Universal Robots PolyScope program: L06_extract_force.urp

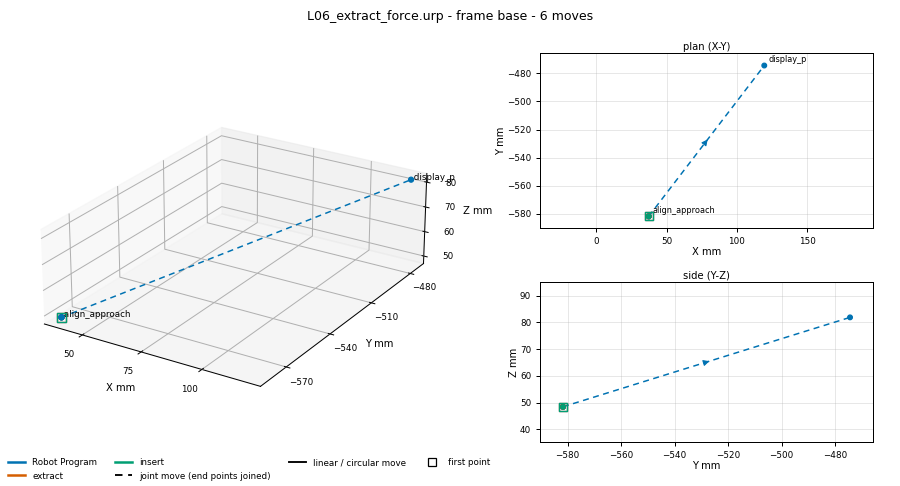
[picture p0: tool path of L06_extract_force.urp in frame base, 6 of 8 moves have a stored position in this frame; points joined in program order, loops and branches not executed]
Program L06_extract_force (installation=default directory=/programs createdIn=5.9.1.1031110 lastSavedIn=5.9.1.1031110 robotSerialNumber=20195501059)
Calibrated DH parameters: a=[0.000146, -0.418764, -0.053981, 0.000058, -0.000023, 0]; d=[0.162545, 37.319448, -206.067439, 168.881546, 0.09955, 0.099464]; alpha=[1.57004, -0.001979, 0.002304, 1.570607, -1.57066, 0]; deltaTheta=[0, -0.174616, -1.258233, 1.432844, -0.000001, 0]
BeforeStart
  URCap Gripper Activate (Robotiq_Grippers, Robotiq Inc.) dataModel(ResetAndActivateKey=false)
  URCap Gripper (Robotiq_Grippers, Robotiq Inc.) dataModel(position=60.0, force=10.0, speed=40.0, positionInDouble=60.0, forceInDouble=10.0, speedInDouble=40.0, slaveIds=[9], blocking=true)
  start_p := get_actual_tcp_pose()
  MoveJ speed 60 deg/s, acceleration 80 deg/s^2 (useActiveTCP=true) feature=Base
    Waypoint Waypoint (Variable): variable=start_p
  MoveL speed 250 mm/s, acceleration 1200 mm/s^2 (useActiveTCP=true) feature=Base
    MoveDirectionNode (selectedDirection=ZPlus)
      Until DISTANCE (allowActions=false deceleration=3 distanceNodeType=STOP) Distance=0.025; motionParameters(blendRadius=0)
  URCap Gripper (Robotiq_Grippers, Robotiq Inc.) dataModel(position=100.0, force=25.0, speed=100.0, positionInDouble=100.0, forceInDouble=25.0, speedInDouble=100.0, slaveIds=[9], blocking=true)
Robot Program (runOnlyOnce=true)
  MoveJ speed 60 deg/s, acceleration 80 deg/s^2 (useActiveTCP=true) feature=Base
    Waypoint align_approach: TCP in base x=37.324 y=-581.757 z=48.473 mm, rx=2.21 ry=2.2328 rz=0 rad; joints [80.399, -68.66, 105.716, -127.049, 270.027, 79.839] deg; TCP offset x=0 y=0 z=174 mm, rx=0 ry=0 rz=0 rad
  MoveL speed 250 mm/s, acceleration 1200 mm/s^2 (useActiveTCP=true) feature=Base
    Waypoint misalign: TCP in base x=37.345 y=-581.767 z=48.476 mm, rx=2.3536 ry=2.027 rz=0.0112 rad; joints [79.512, -69.245, 106.923, -128.62, 271.871, 88.086] deg
    'Touch plug'
    URCap Gripper (Robotiq_Grippers, Robotiq Inc.) dataModel(position=100.0, force=25.0, speed=100.0, positionInDouble=100.0, forceInDouble=25.0, speedInDouble=100.0, slaveIds=[9], blocking=true)
    MoveDirectionNode (selectedDirection=ZPlus toolParams=0.02, 0.8) feature=Joint_6_name
      Until DISTANCE (allowActions=true deceleration=3 distanceNodeType=STOP) Distance=0.025; motionParameters(blendRadius=0)
        MoveL speed 250 mm/s, acceleration 1200 mm/s^2 (useActiveTCP=true) feature=Base
          Waypoint align_approach: TCP in base x=37.324 y=-581.757 z=48.473 mm, rx=2.21 ry=2.2328 rz=0 rad; joints [80.399, -68.66, 105.716, -127.049, 270.027, 79.839] deg
          Halt
      Until TOOL_CONTACT_DETECTION (allowActions=false retraction=0.002 decelerationAcceleration=0.8 decelerationAngularAcceleration=34.906585)
    Call extract
    extract_p := get_actual_tcp_pose()
    MoveDirectionNode (selectedDirection=YPlus) feature=Base
      Until DISTANCE (allowActions=false deceleration=3 distanceNodeType=STOP) Distance=0.05; motionParameters(blendRadius=0)
    MoveJ speed 60 deg/s, acceleration 80 deg/s^2 (useActiveTCP=true) feature=Base
      Waypoint display_p: TCP in base x=119.536 y=-474.453 z=81.895 mm, rx=0.3577 ry=2.5974 rz=0.0553 rad; joints [71.361, -83.619, 123.353, -121.111, 298.741, -5.14] deg
      Wait Sleep waitTime=2
      Waypoint Waypoint (Variable): variable=extract_p
    'Deliberately misalign'
    MoveDirectionNode (selectedDirection=ZPlus) feature=Joint_6_name
      Until DISTANCE (allowActions=false deceleration=3 distanceNodeType=STOP) Distance=0.001; motionParameters(blendRadius=0)
    MoveDirectionNode (selectedDirection=XPlus) feature=Joint_6_name
      Until DISTANCE (allowActions=false deceleration=3 distanceNodeType=STOP) Distance=0.001; motionParameters(blendRadius=0)
    Call insert
SubProgram -> insert
SubProgram -> extract
SubProgram extract (keepSynchronizedWithDisk=false)
  MoveL speed 250 mm/s, acceleration 1200 mm/s^2 (useActiveTCP=true) feature=Base
    URCap Gripper (Robotiq_Grippers, Robotiq Inc.) dataModel(position=60.0, force=100.0, speed=100.0, positionInDouble=60.0, forceInDouble=100.0, speedInDouble=100.0, slaveIds=[9], blocking=true)
    MoveDirectionNode (selectedDirection=ZMinus)
      Until DISTANCE (allowActions=false deceleration=3 distanceNodeType=STOP) Distance=0.02; motionParameters(blendRadius=0)
    URCap Zero FT Sensor (Robotiq_Copilot, Robotiq Inc.) dataModel(NodeInitializedKey=true, WaitForSteadyWrenchOptionKey=true)
    URCap Gripper (Robotiq_Grippers, Robotiq Inc.) dataModel(position=100.0, force=25.0, speed=100.0, positionInDouble=100.0, forceInDouble=25.0, speedInDouble=100.0, slaveIds=[9], blocking=true)
    URCap Grip Check (Robotiq_Grippers, Robotiq Inc.) dataModel(ObjectDetectedKey=true, DimensionValidationKey=false, DimensionKey=100.0, DimensionDimensionPositiveGapKey=5.0, DimensionNegativeGapKey=5.0, GripperIdKey=1, ModelDefinedKey=true); state(isChildrenLocked=true)
      URCap If (Robotiq_Grippers, Robotiq Inc.)
        'plug grabbed'
      URCap Else (Robotiq_Grippers, Robotiq Inc.)
        'no plug'
        MoveJ speed 60 deg/s, acceleration 80 deg/s^2 (useActiveTCP=true) feature=Base
          Waypoint align_approach: TCP in base x=37.324 y=-581.757 z=48.473 mm, rx=2.21 ry=2.2328 rz=0 rad; joints [80.399, -68.66, 105.716, -127.049, 270.027, 79.839] deg
          Halt
    'Let gripper seek alignment'
    URCap Force Control (Robotiq_Copilot, Robotiq Inc.) dataModel(NodeInitializedKey=true, force_x=0, force_y=0, force_z=0, force_mx=0, force_my=0, force_mz=0, limit_x_neg=-100, limit_y_neg=-100, limit_z_neg=-100, limit_x_pos=100, limit_y_pos=100, limit_z_pos=100, limit_mx_neg=-20, limit_my_neg=-20, limit_mz_neg=-20, limit_mx_pos=20, limit_my_pos=20, limit_mz_pos=20, stiffness_x=100, stiffness_y=100, stiffness_z_position=100, stiffness_mx=100, stiffness_my=100, stiffness_mz=100, ft_control_x=true, adaptive_stiffness=true, ft_control_y=true, ft_control_z=true, ft_control_mx=true, ft_control_my=true, ft_control_mz=true, is_force_control_about_actual_position=true, TranslatableFeatureKey=1, HackTriggeringContributionIsDefinedMethodKey=true)
      Wait Sleep waitTime=3
    'Extract'
    URCap Insertion (Robotiq_Copilot, Robotiq Inc.) dataModel(NodeInitializedKey=true)
      URCap Zero FT Sensor (Robotiq_Copilot, Robotiq Inc.) dataModel(NodeInitializedKey=true, WaitForSteadyWrenchOptionKey=false)
      URCap Linear (Robotiq_Copilot, Robotiq Inc.) dataModel(NodeInitializedKey=true, fb_exit_insertion=false, fb_force=40.0, fb_max_distance=40.0, fb_speed=10.0, fbDirection=X+); state(isChildrenLocked=true)
        URCap On error (Robotiq_Copilot, Robotiq Inc.)
          'Sequence if maximum distance is reached'
    SuppressedNode
      URCap Force Control (Robotiq_Copilot, Robotiq Inc.) dataModel(NodeInitializedKey=true, force_z=0, force_mx=0, force_my=0, force_mz=0, limit_x_neg=-100, limit_y_neg=-100, limit_z_neg=-100, limit_x_pos=100, limit_y_pos=100, limit_z_pos=100, limit_mx_neg=-20, limit_my_neg=-20, limit_mz_neg=-20, limit_mx_pos=20, limit_my_pos=20, limit_mz_pos=20, stiffness_x=100, stiffness_y=100, stiffness_z_position=100, stiffness_mx=100, stiffness_my=100, stiffness_mz=100, adaptive_stiffness=true, is_force_control_about_actual_position=true, ft_control_x=true, force_y=0, force_x=40, ft_control_y=true, ft_control_z=true, ft_control_mx=true, ft_control_my=true, ft_control_mz=true, HackTriggeringContributionIsDefinedMethodKey=true, TranslatableFeatureKey=1)
        Wait Sleep waitTime=3
SubProgram insert (keepSynchronizedWithDisk=false)
  URCap Insertion (Robotiq_Copilot, Robotiq Inc.) dataModel(NodeInitializedKey=true)
    URCap Zero FT Sensor (Robotiq_Copilot, Robotiq Inc.) dataModel(NodeInitializedKey=true, WaitForSteadyWrenchOptionKey=true)
    URCap Force Control (Robotiq_Copilot, Robotiq Inc.) dataModel(NodeInitializedKey=true, force_z=0, force_mx=0, force_my=0, force_mz=0, limit_x_neg=-100, limit_y_neg=-100, limit_z_neg=-100, limit_x_pos=100, limit_y_pos=100, limit_z_pos=100, limit_mx_neg=-20, limit_my_neg=-20, limit_mz_neg=-20, limit_mx_pos=20, limit_my_pos=20, limit_mz_pos=20, stiffness_y=100, stiffness_z_position=100, stiffness_mx=100, stiffness_my=100, stiffness_mz=100, adaptive_stiffness=true, is_force_control_about_actual_position=true, ft_control_x=true, force_y=0, stiffness_x=50, ft_control_y=true, ft_control_z=true, ft_control_mx=true, ft_control_my=true, ft_control_mz=true, TranslatableFeatureKey=1, HackTriggeringContributionIsDefinedMethodKey=true, force_x=-20)
      Wait Sleep waitTime=6
    SuppressedNode
      URCap Linear (Robotiq_Copilot, Robotiq Inc.) dataModel(NodeInitializedKey=true, fb_max_distance=100.0, fb_exit_insertion=false, fb_speed=10.0, fb_force=40.0, fbDirection=X-); state(isChildrenLocked=true)
        URCap On error (Robotiq_Copilot, Robotiq Inc.)
          'Sequence if maximum distance is reached'
  URCap Gripper (Robotiq_Grippers, Robotiq Inc.) dataModel(position=60.0, force=25.0, speed=100.0, positionInDouble=60.0, forceInDouble=25.0, speedInDouble=100.0, slaveIds=[9], blocking=true)
  MoveL speed 250 mm/s, acceleration 1200 mm/s^2 (useActiveTCP=true) feature=Base
    Waypoint align_approach: TCP in base x=37.324 y=-581.757 z=48.473 mm, rx=2.21 ry=2.2328 rz=0 rad; joints [80.399, -68.66, 105.716, -127.049, 270.027, 79.839] deg
